FUNCTION_BLOCK FBMACHINE
VAR_INPUT
END_VAR
VAR_OUTPUT
END_VAR
VAR
END_VAR

END_FUNCTION_BLOCK

(* stored: Version 1.1.0.1, ProductVersion 3.1.4026.18
   POU FBMACHINE: Id {c975d90d-848c-4dc5-b717-6d92fef38257}, SpecialFunc None *)
